DATA_BLOCK "LNK_TestVectors"
{ S7_Optimized_Access := 'FALSE' }
VERSION : 0.1
NON_RETAIN
// GENERATED by gr-contract gen-link (registry hash 16#C3CAA074) - do not edit. 표준 접근 : Lnk_SelfTest 골든 벡터
   STRUCT
      Hello_Val : "LNK_Hello";   //   골든 값 (crates/plc-link vectors, sig 16#BFAD9982)
      Hello_Bin : Array[0..27] of Byte;   //   Hello_Val 의 Serialize 바이트 (28 B)
      Hello_JsonLen : DInt;   //   Hello_Json 엔벨로프 텍스트 길이 (seq 1)
      Hello_Json : Array[0..0] of String[200];   //   엔벨로프 텍스트 (200 자씩)
      Ack_Val : "LNK_Ack";   //   골든 값 (crates/plc-link vectors, sig 16#FF5482FF)
      Ack_Bin : Array[0..47] of Byte;   //   Ack_Val 의 Serialize 바이트 (48 B)
      Ack_JsonLen : DInt;   //   Ack_Json 엔벨로프 텍스트 길이 (seq 1)
      Ack_Json : Array[0..0] of String[200];   //   엔벨로프 텍스트 (200 자씩)
      Fixture_Val : "LNK_Fixture";   //   골든 값 (crates/plc-link vectors, sig 16#EB2E5DE0)
      Fixture_Bin : Array[0..169] of Byte;   //   Fixture_Val 의 Serialize 바이트 (170 B)
      Fixture_JsonLen : DInt;   //   Fixture_Json 엔벨로프 텍스트 길이 (seq 1)
      Fixture_Json : Array[0..3] of String[200];   //   엔벨로프 텍스트 (200 자씩)
      FixtureCmd_Val : "LNK_FixtureSub";   //   골든 값 (crates/plc-link vectors, sig 16#AFBB75A6)
      FixtureCmd_Bin : Array[0..25] of Byte;   //   FixtureCmd_Val 의 Serialize 바이트 (26 B)
      FixtureCmd_JsonLen : DInt;   //   FixtureCmd_Json 엔벨로프 텍스트 길이 (seq 1)
      FixtureCmd_Json : Array[0..0] of String[200];   //   엔벨로프 텍스트 (200 자씩)
      JsonOnly_Val : "LNK_FixtureSub";   //   골든 값 (crates/plc-link vectors, sig 16#AFBB75A6)
      JsonOnly_Bin : Array[0..25] of Byte;   //   JsonOnly_Val 의 Serialize 바이트 (26 B)
      JsonOnly_JsonLen : DInt;   //   JsonOnly_Json 엔벨로프 텍스트 길이 (seq 1)
      JsonOnly_Json : Array[0..0] of String[200];   //   엔벨로프 텍스트 (200 자씩)
   END_STRUCT;


BEGIN
   Hello_Val.Plc := 'S8E0EE3EB';
   Hello_Val.Proto := 231;
   Hello_Val.Formats := 16#A0;
   Hello_Val.RegistryHash := 16#91F3_4ED5;
   Hello_Val.HeartbeatMs := 3319752200;
   Hello_Bin[0] := 16#10;
   Hello_Bin[1] := 16#09;
   Hello_Bin[2] := 16#53;
   Hello_Bin[3] := 16#38;
   Hello_Bin[4] := 16#45;
   Hello_Bin[5] := 16#30;
   Hello_Bin[6] := 16#45;
   Hello_Bin[7] := 16#45;
   Hello_Bin[8] := 16#33;
   Hello_Bin[9] := 16#45;
   Hello_Bin[10] := 16#42;
   Hello_Bin[18] := 16#E7;
   Hello_Bin[19] := 16#A0;
   Hello_Bin[20] := 16#91;
   Hello_Bin[21] := 16#F3;
   Hello_Bin[22] := 16#4E;
   Hello_Bin[23] := 16#D5;
   Hello_Bin[24] := 16#C5;
   Hello_Bin[25] := 16#DF;
   Hello_Bin[26] := 16#66;
   Hello_Bin[27] := 16#08;
   Hello_JsonLen := 145;
   Hello_Json[0] := '{"type":"Hello","seq":1,"sig":3215825282,"data":{"Plc":"S8E0EE3EB","Proto":231,"Formats":160,"RegistryHash":2448641749,"HeartbeatMs":3319752200}}';
   Ack_Val.RefType := 7407;
   Ack_Val.RefSeq := 5660;
   Ack_Val.Code := 8102;
   Ack_Val.Text := 'S9BB908F9';
   Ack_Bin[0] := 16#1C;
   Ack_Bin[1] := 16#EF;
   Ack_Bin[2] := 16#16;
   Ack_Bin[3] := 16#1C;
   Ack_Bin[4] := 16#1F;
   Ack_Bin[5] := 16#A6;
   Ack_Bin[6] := 16#28;
   Ack_Bin[7] := 16#09;
   Ack_Bin[8] := 16#53;
   Ack_Bin[9] := 16#39;
   Ack_Bin[10] := 16#42;
   Ack_Bin[11] := 16#42;
   Ack_Bin[12] := 16#39;
   Ack_Bin[13] := 16#30;
   Ack_Bin[14] := 16#38;
   Ack_Bin[15] := 16#46;
   Ack_Bin[16] := 16#39;
   Ack_JsonLen := 108;
   Ack_Json[0] := '{"type":"Ack","seq":1,"sig":4283728639,"data":{"RefType":7407,"RefSeq":5660,"Code":8102,"Text":"S9BB908F9"}}';
   Fixture_Val.B4 := TRUE;
   Fixture_Val.B5 := TRUE;
   Fixture_Val.B6 := TRUE;
   Fixture_Val.B7 := TRUE;
   Fixture_Val."By" := 16#E0;
   Fixture_Val.Si := 20;
   Fixture_Val.I := -26951;
   Fixture_Val.W := 16#2BDA;
   Fixture_Val.Di := -509460222;
   Fixture_Val.Udi := 2697544214;
   Fixture_Val.R := -8289.25;
   Fixture_Val.Lr := 4705.75;
   Fixture_Val.Li := 1494603010750283776;
   Fixture_Val.Ch := 'V';
   Fixture_Val.Str := 'S64E3E51';
   Fixture_Val.Ts.YEAR := 2026;
   Fixture_Val.Ts.MONTH := 9;
   Fixture_Val.Ts.DAY := 13;
   Fixture_Val.Ts.WEEKDAY := 1;
   Fixture_Val.Ts.HOUR := 10;
   Fixture_Val.Ts.MINUTE := 11;
   Fixture_Val.Ts.SECOND := 12;
   Fixture_Val.Ts.NANOSECOND := 345000000;
   Fixture_Val.Ts := DTL#2026-09-13-10:11:12.345;
   Fixture_Val.Tm := T#-7m_9s_593ms;
   Fixture_Val.Flags[0] := TRUE;
   Fixture_Val.Flags[2] := TRUE;
   Fixture_Val.Axis[1] := 2239.75;
   Fixture_Val.Axis[2] := -2439.75;
   Fixture_Val.Axis[3] := -4840.0;
   Fixture_Val.Grid[1,0] := -22516;
   Fixture_Val.Grid[1,1] := -26291;
   Fixture_Val.Grid[2,0] := -11556;
   Fixture_Val.Grid[2,1] := -7267;
   Fixture_Val.Outer.A := 182;
   Fixture_Val.Outer.Inner.Flag := TRUE;
   Fixture_Val.Outer.Inner.Val := 21445;
   Fixture_Val.Sub.Id := 45354;
   Fixture_Val.Sub.Name := 'SE44';
   Fixture_Val.Sub.Pos[1] := -9905.5;
   Fixture_Val.Sub.Pos[2] := -5204.75;
   Fixture_Val.Sub.Pos[3] := -7988.5;
   Fixture_Val.Sub.Pos[4] := -253.25;
   Fixture_Val.Subs[0].Id := 5117;
   Fixture_Val.Subs[0].Name := 'S12E';
   Fixture_Val.Subs[0].On := TRUE;
   Fixture_Val.Subs[0].Pos[1] := 3793.75;
   Fixture_Val.Subs[0].Pos[2] := 4217.75;
   Fixture_Val.Subs[0].Pos[3] := -1561.5;
   Fixture_Val.Subs[0].Pos[4] := 787.0;
   Fixture_Val.Subs[1].Id := 14925;
   Fixture_Val.Subs[1].Name := 'SB49';
   Fixture_Val.Subs[1].On := TRUE;
   Fixture_Val.Subs[1].Pos[1] := 7965.0;
   Fixture_Val.Subs[1].Pos[2] := 4216.75;
   Fixture_Val.Subs[1].Pos[3] := 2245.0;
   Fixture_Val.Subs[1].Pos[4] := -8519.75;
   Fixture_Bin[0] := 16#F0;
   Fixture_Bin[2] := 16#E0;
   Fixture_Bin[3] := 16#14;
   Fixture_Bin[4] := 16#96;
   Fixture_Bin[5] := 16#B9;
   Fixture_Bin[6] := 16#2B;
   Fixture_Bin[7] := 16#DA;
   Fixture_Bin[8] := 16#E1;
   Fixture_Bin[9] := 16#A2;
   Fixture_Bin[10] := 16#41;
   Fixture_Bin[11] := 16#02;
   Fixture_Bin[12] := 16#A0;
   Fixture_Bin[13] := 16#C9;
   Fixture_Bin[14] := 16#42;
   Fixture_Bin[15] := 16#16;
   Fixture_Bin[16] := 16#C6;
   Fixture_Bin[17] := 16#01;
   Fixture_Bin[18] := 16#85;
   Fixture_Bin[20] := 16#40;
   Fixture_Bin[21] := 16#B2;
   Fixture_Bin[22] := 16#61;
   Fixture_Bin[23] := 16#C0;
   Fixture_Bin[28] := 16#14;
   Fixture_Bin[29] := 16#BD;
   Fixture_Bin[30] := 16#E5;
   Fixture_Bin[31] := 16#85;
   Fixture_Bin[36] := 16#56;
   Fixture_Bin[38] := 16#08;
   Fixture_Bin[39] := 16#08;
   Fixture_Bin[40] := 16#53;
   Fixture_Bin[41] := 16#36;
   Fixture_Bin[42] := 16#34;
   Fixture_Bin[43] := 16#45;
   Fixture_Bin[44] := 16#33;
   Fixture_Bin[45] := 16#45;
   Fixture_Bin[46] := 16#35;
   Fixture_Bin[47] := 16#31;
   Fixture_Bin[48] := 16#07;
   Fixture_Bin[49] := 16#EA;
   Fixture_Bin[50] := 16#09;
   Fixture_Bin[51] := 16#0D;
   Fixture_Bin[52] := 16#01;
   Fixture_Bin[53] := 16#0A;
   Fixture_Bin[54] := 16#0B;
   Fixture_Bin[55] := 16#0C;
   Fixture_Bin[56] := 16#14;
   Fixture_Bin[57] := 16#90;
   Fixture_Bin[58] := 16#48;
   Fixture_Bin[59] := 16#40;
   Fixture_Bin[60] := 16#FF;
   Fixture_Bin[61] := 16#F9;
   Fixture_Bin[62] := 16#71;
   Fixture_Bin[63] := 16#E7;
   Fixture_Bin[64] := 16#05;
   Fixture_Bin[66] := 16#45;
   Fixture_Bin[67] := 16#0B;
   Fixture_Bin[68] := 16#FC;
   Fixture_Bin[70] := 16#C5;
   Fixture_Bin[71] := 16#18;
   Fixture_Bin[72] := 16#7C;
   Fixture_Bin[74] := 16#C5;
   Fixture_Bin[75] := 16#97;
   Fixture_Bin[76] := 16#40;
   Fixture_Bin[78] := 16#A8;
   Fixture_Bin[79] := 16#0C;
   Fixture_Bin[80] := 16#99;
   Fixture_Bin[81] := 16#4D;
   Fixture_Bin[82] := 16#D2;
   Fixture_Bin[83] := 16#DC;
   Fixture_Bin[84] := 16#E3;
   Fixture_Bin[85] := 16#9D;
   Fixture_Bin[86] := 16#B6;
   Fixture_Bin[88] := 16#01;
   Fixture_Bin[90] := 16#53;
   Fixture_Bin[91] := 16#C5;
   Fixture_Bin[92] := 16#B1;
   Fixture_Bin[93] := 16#2A;
   Fixture_Bin[94] := 16#04;
   Fixture_Bin[95] := 16#04;
   Fixture_Bin[96] := 16#53;
   Fixture_Bin[97] := 16#45;
   Fixture_Bin[98] := 16#34;
   Fixture_Bin[99] := 16#34;
   Fixture_Bin[102] := 16#C6;
   Fixture_Bin[103] := 16#1A;
   Fixture_Bin[104] := 16#C6;
   Fixture_Bin[106] := 16#C5;
   Fixture_Bin[107] := 16#A2;
   Fixture_Bin[108] := 16#A6;
   Fixture_Bin[110] := 16#C5;
   Fixture_Bin[111] := 16#F9;
   Fixture_Bin[112] := 16#A4;
   Fixture_Bin[114] := 16#C3;
   Fixture_Bin[115] := 16#7D;
   Fixture_Bin[116] := 16#40;
   Fixture_Bin[118] := 16#13;
   Fixture_Bin[119] := 16#FD;
   Fixture_Bin[120] := 16#04;
   Fixture_Bin[121] := 16#04;
   Fixture_Bin[122] := 16#53;
   Fixture_Bin[123] := 16#31;
   Fixture_Bin[124] := 16#32;
   Fixture_Bin[125] := 16#45;
   Fixture_Bin[126] := 16#01;
   Fixture_Bin[128] := 16#45;
   Fixture_Bin[129] := 16#6D;
   Fixture_Bin[130] := 16#1C;
   Fixture_Bin[132] := 16#45;
   Fixture_Bin[133] := 16#83;
   Fixture_Bin[134] := 16#CE;
   Fixture_Bin[136] := 16#C4;
   Fixture_Bin[137] := 16#C3;
   Fixture_Bin[138] := 16#30;
   Fixture_Bin[140] := 16#44;
   Fixture_Bin[141] := 16#44;
   Fixture_Bin[142] := 16#C0;
   Fixture_Bin[144] := 16#3A;
   Fixture_Bin[145] := 16#4D;
   Fixture_Bin[146] := 16#04;
   Fixture_Bin[147] := 16#04;
   Fixture_Bin[148] := 16#53;
   Fixture_Bin[149] := 16#42;
   Fixture_Bin[150] := 16#34;
   Fixture_Bin[151] := 16#39;
   Fixture_Bin[152] := 16#01;
   Fixture_Bin[154] := 16#45;
   Fixture_Bin[155] := 16#F8;
   Fixture_Bin[156] := 16#E8;
   Fixture_Bin[158] := 16#45;
   Fixture_Bin[159] := 16#83;
   Fixture_Bin[160] := 16#C6;
   Fixture_Bin[162] := 16#45;
   Fixture_Bin[163] := 16#0C;
   Fixture_Bin[164] := 16#50;
   Fixture_Bin[166] := 16#C6;
   Fixture_Bin[167] := 16#05;
   Fixture_Bin[168] := 16#1F;
   Fixture_JsonLen := 735;
   Fixture_Json[0] := '{"type":"Fixture","seq":1,"sig":3945684448,"data":{"B0":false,"B1":false,"B2":false,"B3":false,"B4":true,"B5":true,"B6":true,"B7":true,"B8":false,"By":224,"Si":20,"I":-26951,"W":11226,"Di":-509460222,';
   Fixture_Json[1] := '"Udi":2697544214,"R":-8289.25,"Lr":4705.75,"Li":1494603010750283776,"Ch":"V","Str":"S64E3E51","Ts":"2026-09-13T10:11:12.345","Tm":-429593,"Flags":[true,false,true],"Axis":[2239.75,-2439.75,-4840.0],"G';
   Fixture_Json[2] := 'rid":[[-22516,-26291],[-11556,-7267]],"Outer":{"A":182,"Inner":{"Flag":true,"Val":21445}},"Sub":{"Id":45354,"Name":"SE44","On":false,"Pos":[-9905.5,-5204.75,-7988.5,-253.25]},"Subs":[{"Id":5117,"Name"';
   Fixture_Json[3] := ':"S12E","On":true,"Pos":[3793.75,4217.75,-1561.5,787.0]},{"Id":14925,"Name":"SB49","On":true,"Pos":[7965.0,4216.75,2245.0,-8519.75]}]}}';
   FixtureCmd_Val.Id := 17394;
   FixtureCmd_Val.Name := 'SFE1';
   FixtureCmd_Val.Pos[1] := 9772.5;
   FixtureCmd_Val.Pos[2] := 2827.0;
   FixtureCmd_Val.Pos[3] := -8351.5;
   FixtureCmd_Val.Pos[4] := -5468.75;
   FixtureCmd_Bin[0] := 16#43;
   FixtureCmd_Bin[1] := 16#F2;
   FixtureCmd_Bin[2] := 16#04;
   FixtureCmd_Bin[3] := 16#04;
   FixtureCmd_Bin[4] := 16#53;
   FixtureCmd_Bin[5] := 16#46;
   FixtureCmd_Bin[6] := 16#45;
   FixtureCmd_Bin[7] := 16#31;
   FixtureCmd_Bin[10] := 16#46;
   FixtureCmd_Bin[11] := 16#18;
   FixtureCmd_Bin[12] := 16#B2;
   FixtureCmd_Bin[14] := 16#45;
   FixtureCmd_Bin[15] := 16#30;
   FixtureCmd_Bin[16] := 16#B0;
   FixtureCmd_Bin[18] := 16#C6;
   FixtureCmd_Bin[19] := 16#02;
   FixtureCmd_Bin[20] := 16#7E;
   FixtureCmd_Bin[22] := 16#C5;
   FixtureCmd_Bin[23] := 16#AA;
   FixtureCmd_Bin[24] := 16#E6;
   FixtureCmd_JsonLen := 130;
   FixtureCmd_Json[0] := '{"type":"FixtureCmd","seq":1,"sig":2948298150,"data":{"Id":17394,"Name":"SFE1","On":false,"Pos":[9772.5,2827.0,-8351.5,-5468.75]}}';
   JsonOnly_Val.Id := 17394;
   JsonOnly_Val.Name := 'SFE1';
   JsonOnly_Val.Pos[1] := 9772.5;
   JsonOnly_Val.Pos[2] := 2827.0;
   JsonOnly_Val.Pos[3] := -8351.5;
   JsonOnly_Val.Pos[4] := -5468.75;
   JsonOnly_Bin[0] := 16#43;
   JsonOnly_Bin[1] := 16#F2;
   JsonOnly_Bin[2] := 16#04;
   JsonOnly_Bin[3] := 16#04;
   JsonOnly_Bin[4] := 16#53;
   JsonOnly_Bin[5] := 16#46;
   JsonOnly_Bin[6] := 16#45;
   JsonOnly_Bin[7] := 16#31;
   JsonOnly_Bin[10] := 16#46;
   JsonOnly_Bin[11] := 16#18;
   JsonOnly_Bin[12] := 16#B2;
   JsonOnly_Bin[14] := 16#45;
   JsonOnly_Bin[15] := 16#30;
   JsonOnly_Bin[16] := 16#B0;
   JsonOnly_Bin[18] := 16#C6;
   JsonOnly_Bin[19] := 16#02;
   JsonOnly_Bin[20] := 16#7E;
   JsonOnly_Bin[22] := 16#C5;
   JsonOnly_Bin[23] := 16#AA;
   JsonOnly_Bin[24] := 16#E6;
   JsonOnly_JsonLen := 128;
   JsonOnly_Json[0] := '{"type":"JsonOnly","seq":1,"sig":2948298150,"data":{"Id":17394,"Name":"SFE1","On":false,"Pos":[9772.5,2827.0,-8351.5,-5468.75]}}';

END_DATA_BLOCK
